(* PLC project Beremiz wxHMI test, beremiz Beremiz 0.0 *)
(* stored: creationDateTime 2008-12-14T16:21:19, modificationDateTime 2017-06-05T14:01:40 *)

PROGRAM main_pytest
  VAR
    getCheckBoxState : python_poll;
    counter : INT;
    setSpinCtrlValue : python_poll;
  END_VAR
  VAR  (* added by the conversion: wires and edge detectors of the diagram *)
    _STRING_TO_INT30_ENO : BOOL;
    _STRING_TO_INT30_OUT : INT;
    _ADD32_ENO : BOOL;
    _ADD32_OUT : INT;
    _INT_TO_STRING35_ENO : BOOL;
    _INT_TO_STRING35_OUT : STRING;
    _CONCAT34_ENO : BOOL;
    _CONCAT34_OUT : STRING;
  END_VAR

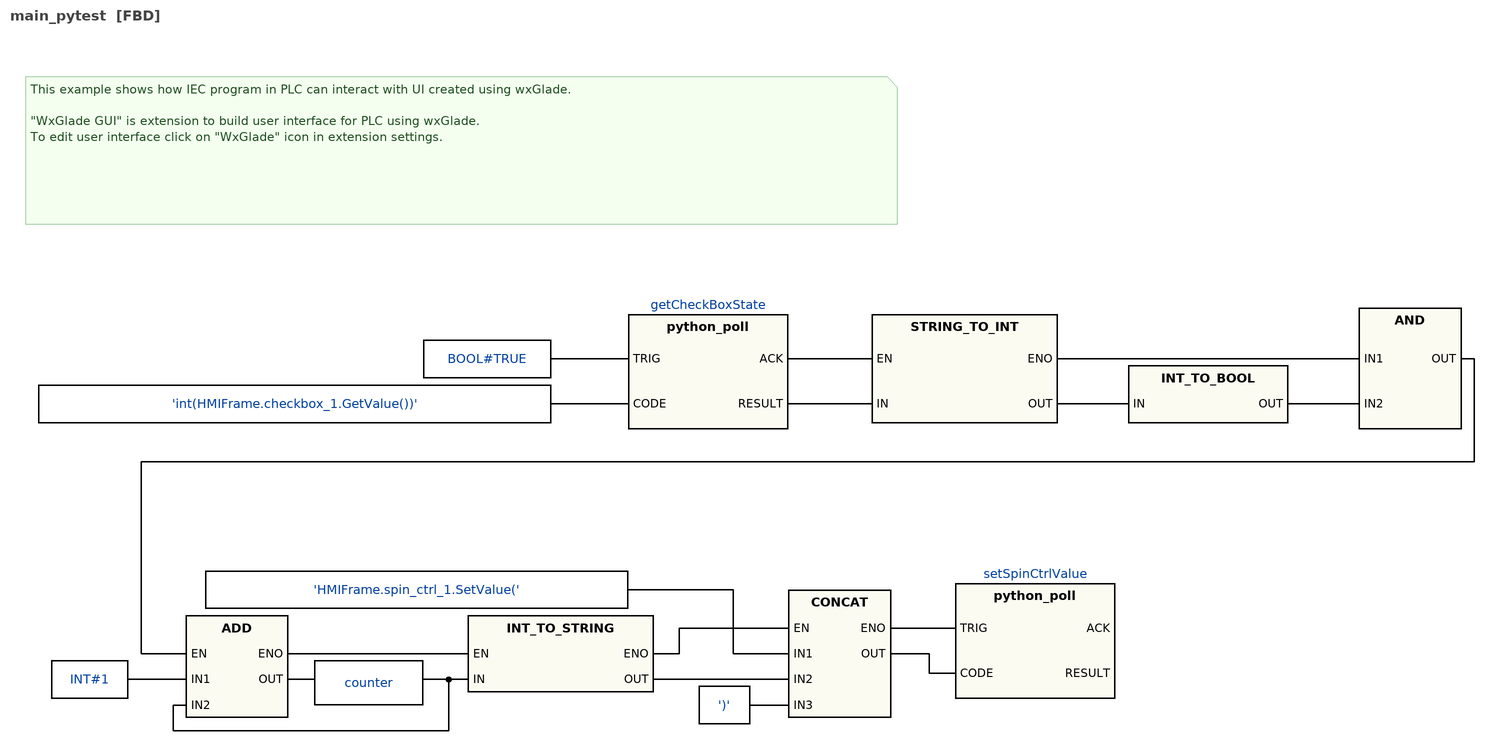
(* FBD diagram, written out as Structured Text *)
(* This example shows how IEC program in PLC can interact with UI created using wxGlade. 

"WxGlade GUI" is extension to build user interface for PLC using wxGlade.
To edit user interface click on "WxGlade" icon in extension settings. *)
getCheckBoxState(TRIG := BOOL#TRUE, CODE := 'int(HMIFrame.checkbox_1.GetValue())');
_STRING_TO_INT30_OUT := STRING_TO_INT(EN := getCheckBoxState.ACK, IN := getCheckBoxState.RESULT, ENO => _STRING_TO_INT30_ENO);
_ADD32_OUT := ADD(EN := _STRING_TO_INT30_ENO AND INT_TO_BOOL(_STRING_TO_INT30_OUT), IN1 := INT#1, IN2 := counter, ENO => _ADD32_ENO);
IF _ADD32_ENO THEN counter := _ADD32_OUT; END_IF;
_INT_TO_STRING35_OUT := INT_TO_STRING(EN := _ADD32_ENO, IN := counter, ENO => _INT_TO_STRING35_ENO);
_CONCAT34_OUT := CONCAT(EN := _INT_TO_STRING35_ENO, IN1 := 'HMIFrame.spin_ctrl_1.SetValue(', IN2 := _INT_TO_STRING35_OUT, IN3 := ')', ENO => _CONCAT34_ENO);
setSpinCtrlValue(TRIG := _CONCAT34_ENO, CODE := _CONCAT34_OUT);
END_PROGRAM

CONFIGURATION config
  RESOURCE res_pytest ON PLC
    TASK pytest_task(INTERVAL := t#100ms, PRIORITY := 0);
    PROGRAM pytest_instance : main_pytest;
  END_RESOURCE
END_CONFIGURATION
